(* IEC 61131-3 sources: AxTestProject/Program/Untitled, 2 files *)

(* ---- Configuration.st ---- *)
CONFIGURATION PLC_1

    var_global
        sysLibTimer : DINT;

        DI_0_0 AT %I0.0 : BOOL;
        DQ_0_0 AT %Q0.0 : BOOL;
        DQ_0_1 AT %Q0.1 : BOOL;
        DQ_0_2 AT %Q0.1 : BOOL;

        S100 : stdLib.SignalHandling.BinSignal;
        H100 : stdLib.SignalHandling.BinOutput;
        Q_M1 : stdLib.SignalHandling.BinOutput;

        PushButton : Application.PushButton;
        Bulb : Application.Bulb;
        M1 : Application.Motor;

        //--------------------------------------------------
        // Programm Light LightStack
        //--------------------------------------------------
        isInitialized : BOOL;
        Signal_0_0 : stdLib.SignalHandling.BinOutput;
        Signal_0_1 : stdLib.SignalHandling.BinOutput;
        Signal_0_2 : stdLib.SignalHandling.BinOutput;

        lampRed : Application.Bulb;
        lampYellow : Application.Bulb;
        lampGreen : Application.Bulb;

        stateINIT : stdLib.Statemachine.State;
        stateRed : stdLib.Statemachine.State;
        stateYellow : stdLib.Statemachine.State;
        stateGreen : stdLib.Statemachine.State;

    end_var

    TASK Main(Priority := 1);
    TASK System(Interval := T#10ms, Priority := 1);

    //PROGRAM P1 WITH Main : TestProgramm;
    PROGRAM PLightStack WITH Main : LightStack;
    PROGRAM P2 WITH System : Timer;

END_CONFIGURATION

(* ---- Timer.st ---- *)
PROGRAM Timer
    VAR_TEMP
    END_VAR
    VAR_EXTERNAL
        sysLibTimer : DINT;
    END_VAR;

    sysLibTimer := (sysLibTimer + DINT#10) MOD System.Const.MaxTimer(); // increment by 10ms --> must be match with the task configuration "interval := 10ms";

END_PROGRAM
